(* LS Electric XG5000 project: XMC_NC_ImportProgram *)
(* example program for importing NC file from SD card. *)
(* PLC LSPLC *)
(* module base 0 slot 0: Input/Output Module:XMC-DN24 (DC 24V Input 8Points/TR output 16Points) *)
(* module base 0 slot 1: Internal Analog Input/Output:XMF-AH04E (A/D voltage/current 2 channels, D/A voltage 2 channels) *)
(* task Periodic Task: Kind=2 *)
(* task Initialization Task: Kind=1 *)
(* task NC Program: Kind=6 *)

PROGRAM NC_Example (* task: Scan Program *)
VAR
    Axes_Busy : BOOL; (* flag to check busy status of NC axes *)
    Axes_On : BOOL; (* flag to check that 3 NC axes are powered on *)
    Axes_Ready : BOOL; (* flag that 3 NC channel axes are ready. *)
    Connect_INST : LS_CONNECT; (* LS_Connect FB *)
    Execute_Connect : BOOL; (* flag to execute LS_Connect FB *)
    Execute_Disconnect : BOOL; (* disconnect the EtherCAT network *)
    Execute_Homing : BOOL; (* flag to home all axes *)
    Execute_ImportProgram : BOOL; (* import NC program from SD memory card *)
    Execute_LoadNCProgram : BOOL; (* flag to load program into NC Channel *)
    Execute_Power : BOOL; (* flag to power on all axes *)
    Execute_StartCycle : BOOL; (* flag to run NC program *)
    INST_CycleStart : NC_CYCLESTART; (* FB to start NC program cycle *)
    INST_Disconnect : LS_DISCONNECT; (* LS_Disconnect FB *)
    INST_HomeAll : MC_HOMEALL; (* FB to home all axes *)
    INST_ImportProgram : NC_IMPORTPROGRAM; (* NC_ImportProgram FB *)
    INST_LoadProgram : NC_LOADPROGRAM; (* FB to load NC program for channel to run *)
    INST_NCReset : NC_RESET; (* FB to reset NC Channel *)
    INST_PowerAll : MC_POWERALL; (* FB to power all servos *)
    NcChannel : UINT := 1; (* NC Channel to perform commands on *)
    resetNC : BOOL; (* flag to reset NC Channel *)
END_VAR

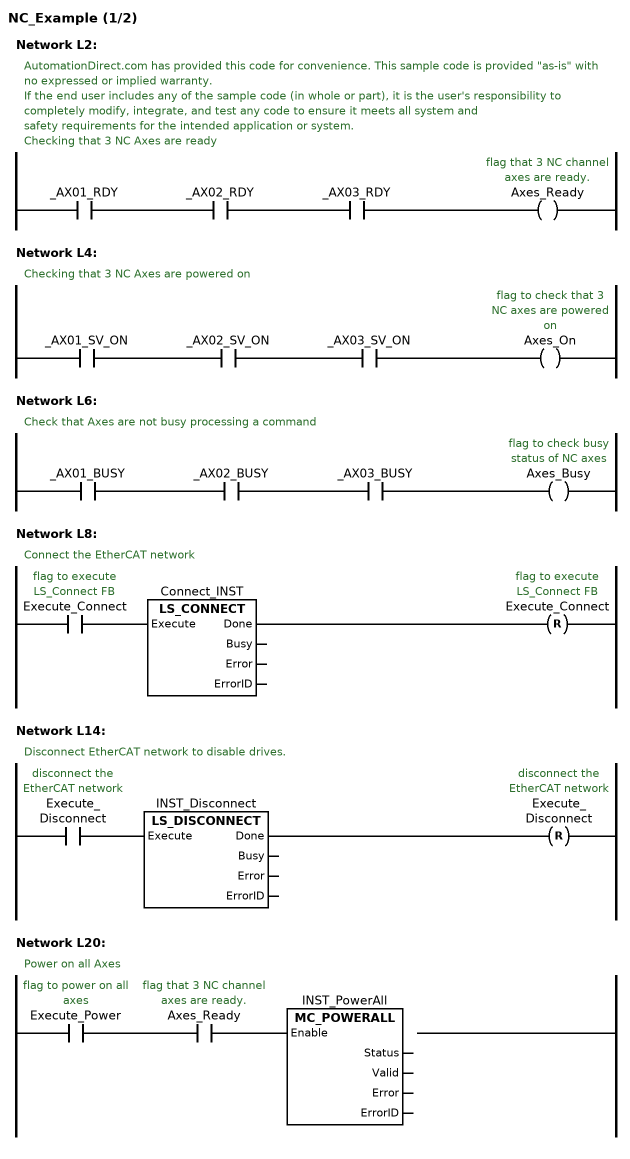
(* AutomationDirect.com has provided this code for convenience. This sample code is provided "as-is" with no expressed or implied warranty. / If the end user includes any of the sample code (in whole or part), it is the user's responsibility to completely modify, integrate, and test any code to ensure it meets all system and / safety requirements for the intended application or system. *)
(* Checking that 3 NC Axes are ready *)
(* Rung L2 *)
Axes_Ready := _AX01_RDY AND _AX02_RDY AND _AX03_RDY;
(* Checking that 3 NC Axes are powered on *)
(* Rung L4 *)
Axes_On := _AX01_SV_ON AND _AX02_SV_ON AND _AX03_SV_ON;
(* Check that Axes are not busy processing a command *)
(* Rung L6 *)
Axes_Busy := _AX01_BUSY AND _AX02_BUSY AND _AX03_BUSY;
(* Connect the EtherCAT network *)
(* Rung L8 *)
Connect_INST(Execute := Execute_Connect);
IF Connect_INST.Done THEN Execute_Connect := FALSE; END_IF;
(* Disconnect EtherCAT network to disable drives. *)
(* Rung L14 *)
INST_Disconnect(Execute := Execute_Disconnect);
IF INST_Disconnect.Done THEN Execute_Disconnect := FALSE; END_IF;
(* Power on all Axes *)
(* Rung L20 *)
INST_PowerAll(Enable := Execute_Power AND Axes_Ready);

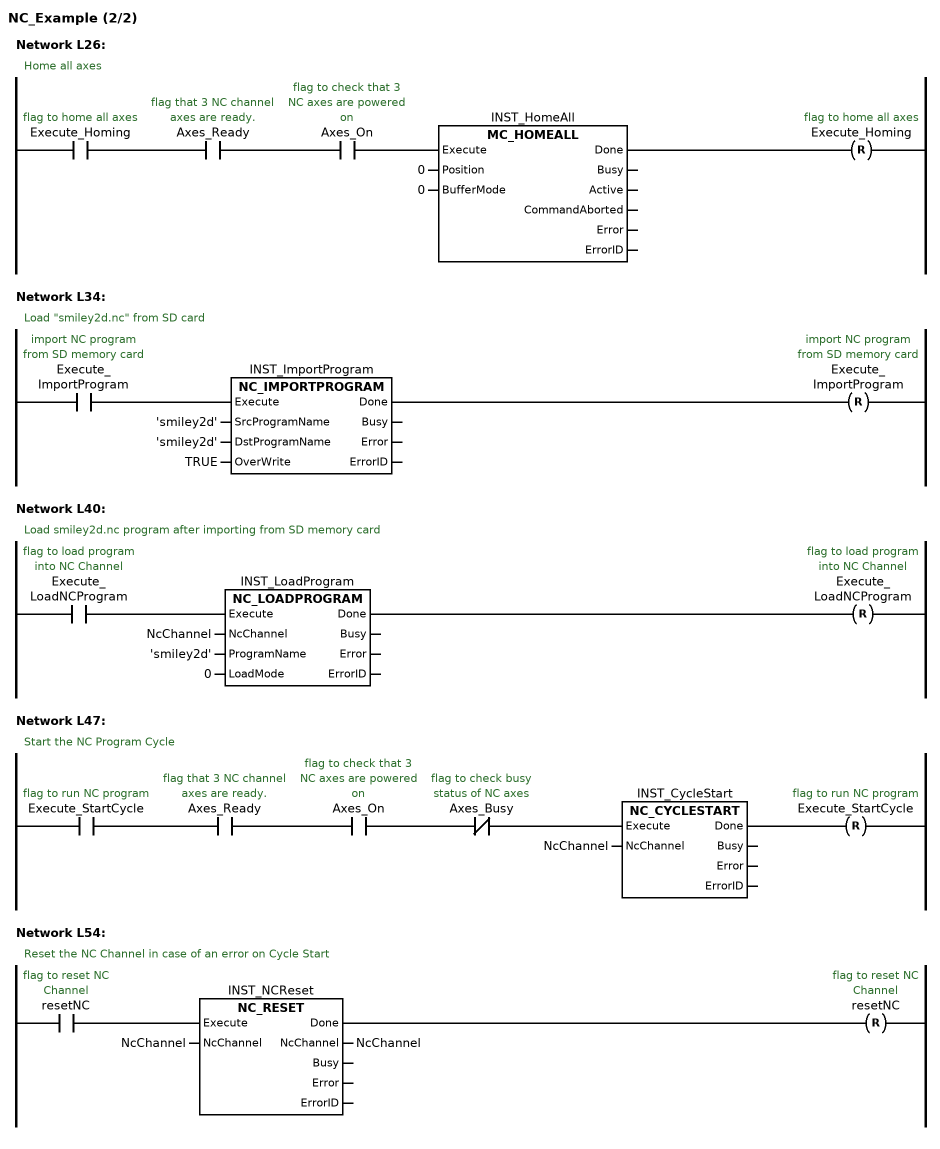
(* Home all axes *)
(* Rung L26 *)
INST_HomeAll(Execute := Execute_Homing AND Axes_Ready AND Axes_On, Position := 0, BufferMode := 0);
IF INST_HomeAll.Done THEN Execute_Homing := FALSE; END_IF;
(* Load "smiley2d.nc" from SD card *)
(* Rung L34 *)
INST_ImportProgram(Execute := Execute_ImportProgram, SrcProgramName := 'smiley2d', DstProgramName := 'smiley2d', OverWrite := TRUE);
IF INST_ImportProgram.Done THEN Execute_ImportProgram := FALSE; END_IF;
(* Load smiley2d.nc program after importing from SD memory card *)
(* Rung L40 *)
INST_LoadProgram(Execute := Execute_LoadNCProgram, NcChannel := NcChannel, ProgramName := 'smiley2d', LoadMode := 0);
IF INST_LoadProgram.Done THEN Execute_LoadNCProgram := FALSE; END_IF;
(* Start the NC Program Cycle *)
(* Rung L47 *)
INST_CycleStart(Execute := Execute_StartCycle AND Axes_Ready AND Axes_On AND NOT Axes_Busy, NcChannel := NcChannel);
IF INST_CycleStart.Done THEN Execute_StartCycle := FALSE; END_IF;
(* Reset the NC Channel in case of an error on Cycle Start *)
(* Rung L54 *)
INST_NCReset(Execute := resetNC, NcChannel := NcChannel, NcChannel => NcChannel);
IF INST_NCReset.Done THEN resetNC := FALSE; END_IF;
END_PROGRAM